# B&R Automation Studio project Tmp_Recipe_V1 (part 2)

### Variables.var - not listed in the package file held
```iecst
(*------------------------------------------------------------------------------------------------------------------------------------------------------------------------------------------------------------------------*)
(*Configuration for recipe managment*)
VAR CONSTANT
	REC_USE_UNICODE : BOOL := FALSE; (*Use standard strings for recipe name when false, use unicode strings for recipe name when true*)
	REC_SORT_NUMERIC : BOOL := FALSE; (*Sort recipe names as numeric values instead of alphabetic*)
END_VAR
VAR
	REC_RECIPE_TYPE : recTYPE := typeCSV; (*Type of recipe (CSV / XML)*)
END_VAR
VAR CONSTANT
	REC_MAX_NUM : USINT := 100; (*Maximum number of recipes*)
	REC_UPLOAD_DOWNLOAD_SIZE : UDINT := 100000; (*Maximum size of memory allocated for uploading and downloading files*)
	REC_NAME_LENGTH : USINT := 40; (*Maximum length for a recipe name*)
	REC_VIS_LENGTH : USINT := 120; (*Make this REC_NAME_LENGTH  x3*)
	REC_MAX_CLIENTS_ID : USINT := 2; (*Highest client ID for concurrent web client connections. Do not change this number.*)
END_VAR
VAR
	REC_VIEW_FILTER : ARRAY[0..9] OF STRING[5] := ['csv','xml',8('')]; (*Files extensions than can be used with the view command*)
	Recipe_01 : recMAIN; (*Global recipe structure. The name must match the task name of the recipe managment.*)
	RecipeData : recVariable; (*Structure that contains the recipe variables*)
END_VAR
```

### Program Logical/TestTask

#### Variables.var
```iecst
VAR
	cmd_create : BOOL;
	tmpStr1 : STRING[80];
	tmpStr2 : STRING[80];
	counter : UDINT;
	idx : UINT;
END_VAR
```

#### Main.st
```iecst
PROGRAM _CYCLIC
	// Create sample recipes
	IF(cmd_create AND NOT Recipe_01.CMD.New AND Recipe_01.ERR.No = 0) THEN
		idx := idx + 1;
		MaschineData.Temperature1 := idx;
		MaschineData.Temperature2 := idx;
		MaschineData.Position := idx;
		MaschineData.MotorSpeed := idx;

		brsitoa(idx, ADR(tmpStr1));
		tmpStr2 := 'recipe_';
		brsstrcat(ADR(tmpStr2), ADR(tmpStr1));
		brwcsconv(ADR(Recipe_01.PAR.RecipeName), ADR(tmpStr2), brwU8toUC);
		Recipe_01.CMD.New := 1;

		IF(idx = 100) THEN
			idx := 0;
			cmd_create := FALSE;
		END_IF
	ELSIF (Recipe_01.ERR.No <> 0) THEN
		idx := 0;
		cmd_create := FALSE;
	END_IF

	// Timer for init command
	IF(cmd_create OR Recipe_01.CMD.Init) THEN
		counter := counter + 1;
	END_IF

END_PROGRAM
```

Listed in the project but not available here: Logical/Global.typ, Logical/Global.var
